FUNCTION_BLOCK NodeOfTest EXTENDS Node
VAR_INPUT
END_VAR
VAR_OUTPUT
END_VAR
VAR
END_VAR

{attribute 'monitoring:= 'variable'}
PROPERTY data : STRING
GET
END_GET
SET
END_SET
END_PROPERTY

END_FUNCTION_BLOCK

(* stored: Version 1.1.0.1, ProductVersion 3.1.4024.11
   POU NodeOfTest: Id {e916b9b9-e1bf-4cae-a8c6-1ea565c9be20}, SpecialFunc None
   Property data: Id {8a92affa-770d-4ada-9202-1a21fd11fd5e}
   Get Get: Id {067f7be3-2bac-4463-a192-8f402b2622f3}
   Set Set: Id {5f3f6679-be24-4f9b-beae-0a752a5802fb} *)
